Staubli VAL3: selectAxis.dtx

num nKey = -1
public num nPage = 10
num nRefresh = 498.406
num nTime = 1
num nValue[4]
  [0] = 1
  [1] = 2
  [2] = 3
  [3] = 4
string sDeeperSession
public string sItems
string sMenu[8]
  [0] = "Program Menu"
  [1] = "Trajectory Menu"
  [2] = "Enable laser"
  [3] = "Table frame"
  [4] = "PRODUCTION PAGE"
  [6] = "Advance"
  [7] = "Quit"
string sMenu8[8]
string sMessage
string sPathSession
string sSession
string sVersion = "ValTending 6.1.3.1"
bool bButton[8]
  [0] = true
  [1] = true
  [2] = true
  [3] = true
  [4] = true
  [6] = true
  [7] = true
bool bLaserOn
bool bInterlock
